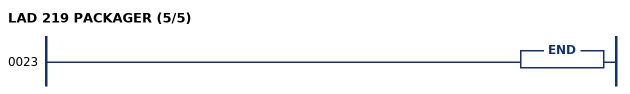
% Rung: 23 %
SOR END EOR

LADDER 220 "NO PACKAGE"
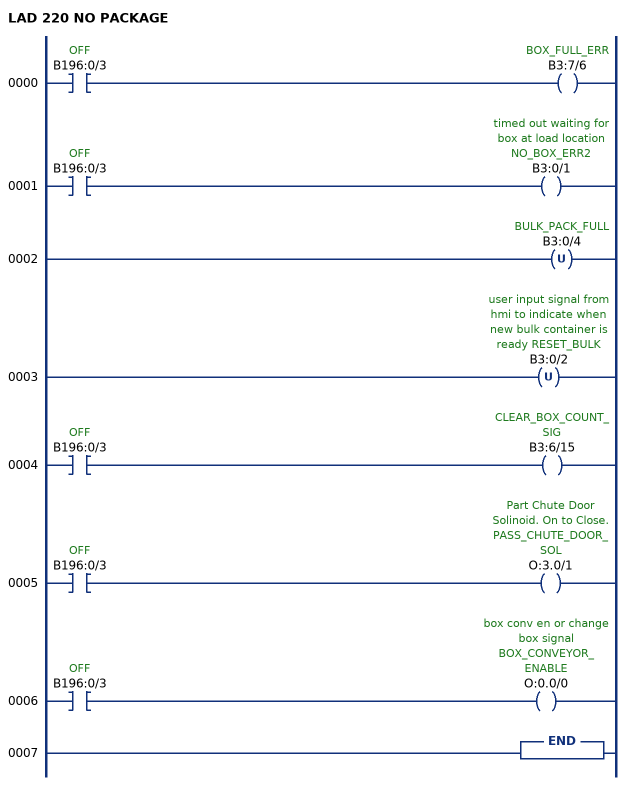
% Rung: 0 %
SOR XIC B196:0/3 OTE B3:7/6 EOR
%   B196:0/3  OFF %
%   B3:7/6  BOX_FULL_ERR %
% Rung: 1 %
SOR XIC B196:0/3 OTE B3:0/1 EOR
%   B196:0/3  OFF %
%   B3:0/1  NO_BOX_ERR2  "timed out waiting for box at load location" %
% Rung: 2 %
SOR OTU B3:0/4 EOR
%   B3:0/4  BULK_PACK_FULL %
% Rung: 3 %
SOR OTU B3:0/2 EOR
%   B3:0/2  RESET_BULK  "user input signal from hmi to indicate when new bulk container is ready" %
% Rung: 4 %
SOR XIC B196:0/3 OTE B3:6/15 EOR
%   B196:0/3  OFF %
%   B3:6/15  CLEAR_BOX_COUNT_SIG %
% Rung: 5 %
SOR XIC B196:0/3 OTE O:3.0/1 EOR
%   B196:0/3  OFF %
%   O:3.0/1  PASS_CHUTE_DOOR_SOL  "Part Chute Door Solinoid. On to Close." %
% Rung: 6 %
SOR XIC B196:0/3 OTE O:0.0/0 EOR
%   B196:0/3  OFF %
%   O:0.0/0  BOX_CONVEYOR_ENABLE  "box conv en or change box signal" %
% Rung: 7 %
SOR END EOR

LADDER 222 "RATE1"
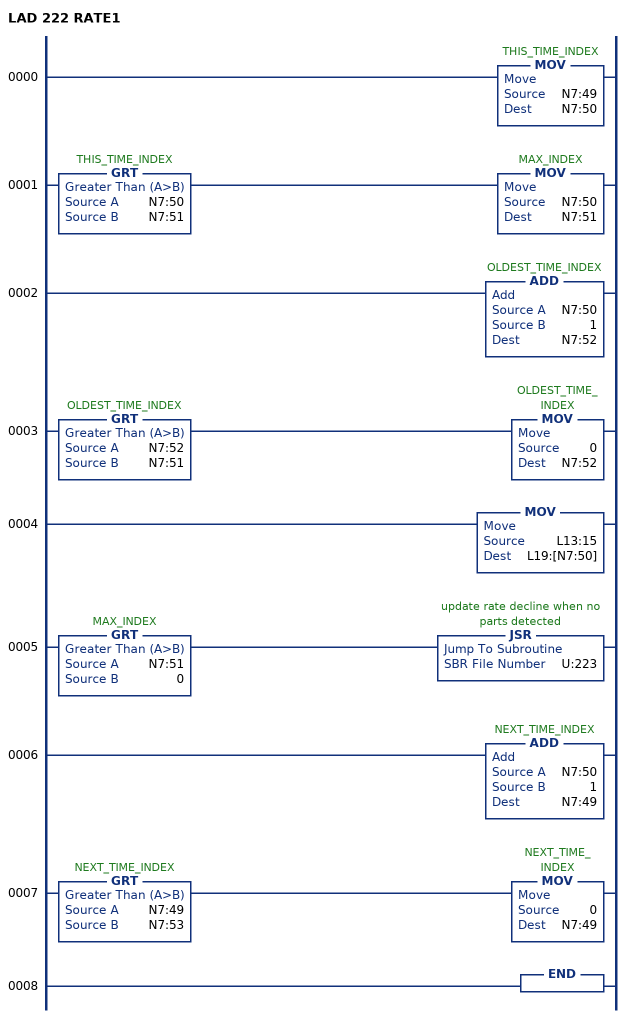
% Rung: 0 %
SOR MOV N7:49 N7:50 EOR
%   N7:49  NEXT_TIME_INDEX %
%   N7:50  THIS_TIME_INDEX %
% Rung: 1 %
SOR GRT N7:50 N7:51 MOV N7:50 N7:51 EOR
%   N7:50  THIS_TIME_INDEX %
%   N7:51  MAX_INDEX %
% Rung: 2 %
SOR ADD N7:50 1 N7:52 EOR
%   N7:50  THIS_TIME_INDEX %
%   N7:52  OLDEST_TIME_INDEX %
% Rung: 3 %
SOR GRT N7:52 N7:51 MOV 0 N7:52 EOR
%   N7:52  OLDEST_TIME_INDEX %
%   N7:51  MAX_INDEX %
% Rung: 4 %
SOR MOV L13:15 L19:[N7:50] EOR
%   L13:15  THE_TIME %
%   N7:50  THIS_TIME_INDEX %
% Rung: 5 %
SOR GRT N7:51 0 JSR U:223 EOR
%   N7:51  MAX_INDEX %
%   U:223  "update rate decline when no parts detected" %
% Rung: 6 %
SOR ADD N7:50 1 N7:49 EOR
%   N7:50  THIS_TIME_INDEX %
%   N7:49  NEXT_TIME_INDEX %
% Rung: 7 %
SOR GRT N7:49 N7:53 MOV 0 N7:49 EOR
%   N7:49  NEXT_TIME_INDEX %
%   N7:53  UPPER_INDEX_LIMIT %
% Rung: 8 %
SOR END EOR

LADDER 223 "RATE2"
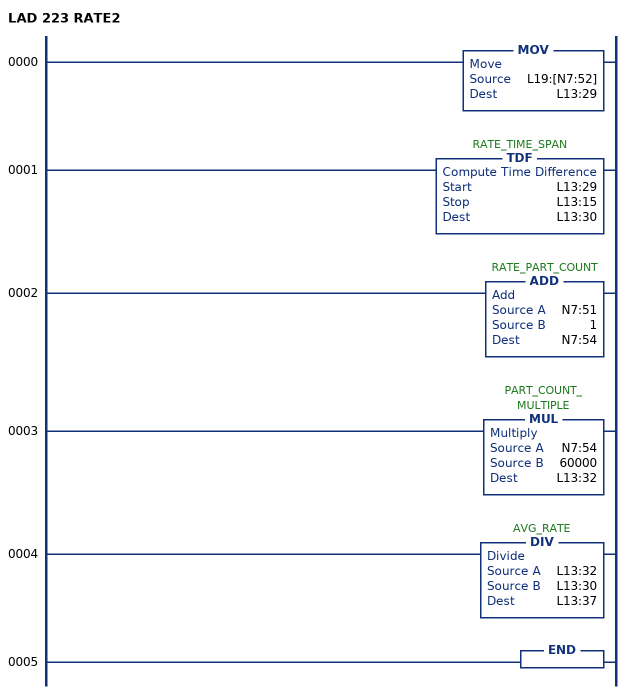
% Rung: 0 %
SOR MOV L19:[N7:52] L13:29 EOR
%   N7:52  OLDEST_TIME_INDEX %
% Rung: 1 %
SOR TDF L13:29 L13:15 L13:30 EOR
%   L13:15  THE_TIME %
%   L13:30  RATE_TIME_SPAN %
% Rung: 2 %
SOR ADD N7:51 1 N7:54 EOR
%   N7:51  MAX_INDEX %
%   N7:54  RATE_PART_COUNT %
% Rung: 3 %
SOR MUL N7:54 60000 L13:32 EOR
%   N7:54  RATE_PART_COUNT %
%   L13:32  PART_COUNT_MULTIPLE %
% Rung: 4 %
SOR DIV L13:32 L13:30 L13:37 EOR
%   L13:32  PART_COUNT_MULTIPLE %
%   L13:30  RATE_TIME_SPAN %
%   L13:37  AVG_RATE %
% Rung: 5 %
SOR END EOR

LADDER 224 "RESET RATE"
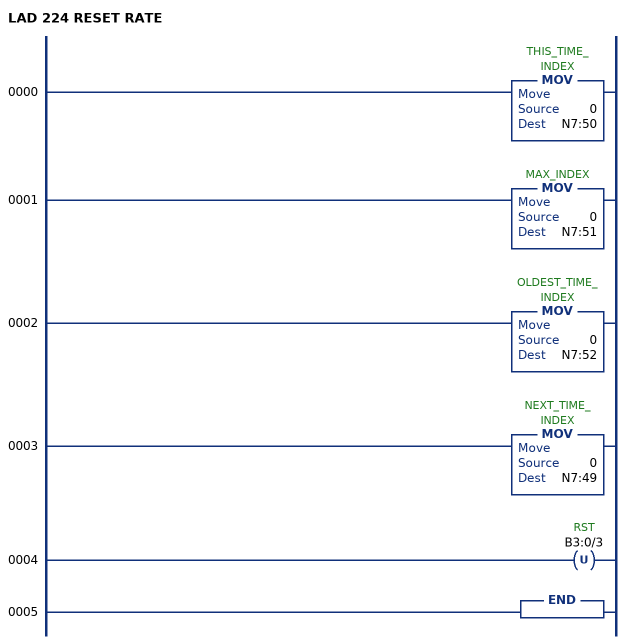
% Rung: 0 %
SOR MOV 0 N7:50 EOR
%   N7:50  THIS_TIME_INDEX %
% Rung: 1 %
SOR MOV 0 N7:51 EOR
%   N7:51  MAX_INDEX %
% Rung: 2 %
SOR MOV 0 N7:52 EOR
%   N7:52  OLDEST_TIME_INDEX %
% Rung: 3 %
SOR MOV 0 N7:49 EOR
%   N7:49  NEXT_TIME_INDEX %
% Rung: 4 %
SOR OTU B3:0/3 EOR
%   B3:0/3  RST %
% Rung: 5 %
SOR END EOR

LADDER 240 "NP STOP"
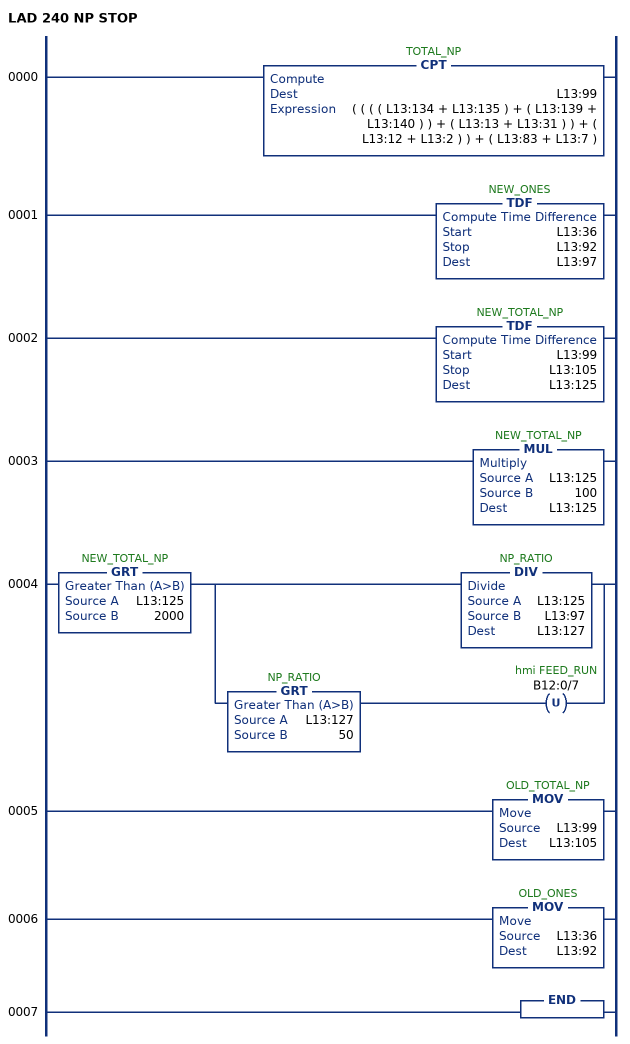
% Rung: 0 %
SOR CPT L13:99 " ( ( ( ( L13:134 + L13:135 ) + ( L13:139 + L13:140 ) ) + ( L13:13 + L13:31 ) ) + ( L13:12 + L13:2 ) ) + ( L13:83 + L13:7 ) " EOR
%   L13:99  TOTAL_NP %
%   L13:134  "too wide bottom" %
%   L13:135  "too close bottom" %
%   L13:139  "too close top count" %
%   L13:140  "too wide top count" %
%   L13:13  SKIP1  "skipped 1 count" %
%   L13:31  SKIP5  "skipped 5 count" %
%   L13:12  SKIP6  "skipped 6 count" %
%   L13:2  INS1_FAIL_COUNT %
%   L13:83  INS5_FAIL_COUNT %
%   L13:7  INS6_FAIL_COUNT %
% Rung: 1 %
SOR TDF L13:36 L13:92 L13:97 EOR
%   L13:36  ONES %
%   L13:92  OLD_ONES %
%   L13:97  NEW_ONES %
% Rung: 2 %
SOR TDF L13:99 L13:105 L13:125 EOR
%   L13:99  TOTAL_NP %
%   L13:105  OLD_TOTAL_NP %
%   L13:125  NEW_TOTAL_NP %
% Rung: 3 %
SOR MUL L13:125 100 L13:125 EOR
%   L13:125  NEW_TOTAL_NP %
% Rung: 4 %
SOR GRT L13:125 2000 BST DIV L13:125 L13:97 L13:127 NXB GRT L13:127 50 OTU B12:0/7 BND EOR
%   L13:125  NEW_TOTAL_NP %
%   L13:97  NEW_ONES %
%   L13:127  NP_RATIO %
%   B12:0/7  FEED_RUN  "hmi" %
% Rung: 5 %
SOR MOV L13:99 L13:105 EOR
%   L13:99  TOTAL_NP %
%   L13:105  OLD_TOTAL_NP %
% Rung: 6 %
SOR MOV L13:36 L13:92 EOR
%   L13:36  ONES %
%   L13:92  OLD_ONES %
% Rung: 7 %
SOR END EOR

LADDER 246 "SPEED BOT"    % high speed %
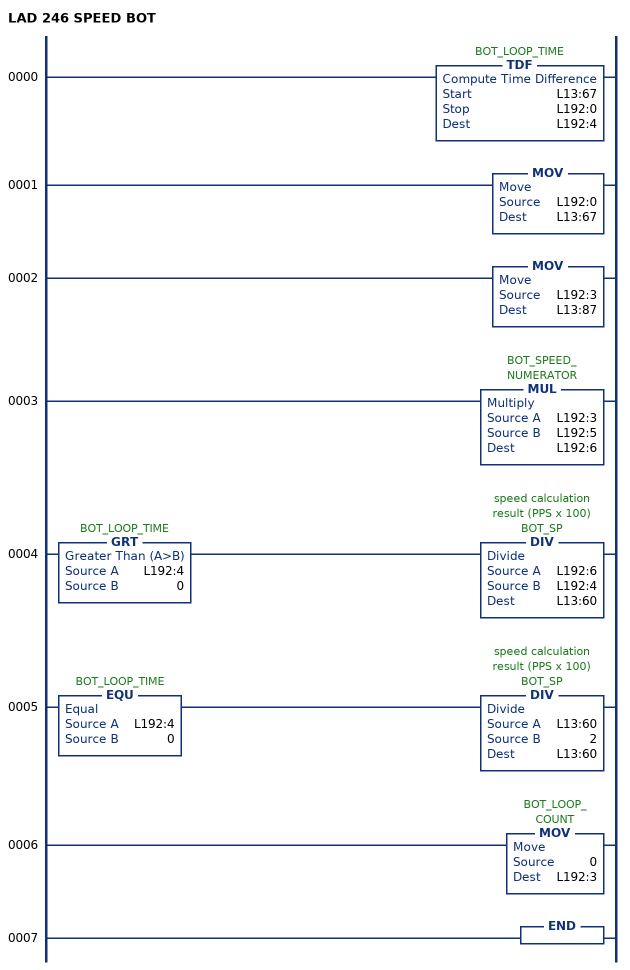
% Rung: 0 %
SOR TDF L13:67 L192:0 L192:4 EOR
%   L192:0  BOT_THIS_TIME  "rtc bot belt movement event time" %
%   L192:4  BOT_LOOP_TIME %
% Rung: 1 %
SOR MOV L192:0 L13:67 EOR
%   L192:0  BOT_THIS_TIME  "rtc bot belt movement event time" %
% Rung: 2 %
SOR MOV L192:3 L13:87 EOR
%   L192:3  BOT_LOOP_COUNT %
% Rung: 3 %
SOR MUL L192:3 L192:5 L192:6 EOR
%   L192:3  BOT_LOOP_COUNT %
%   L192:5  TKS_PER_SECOND %
%   L192:6  BOT_SPEED_NUMERATOR %
% Rung: 4 %
SOR GRT L192:4 0 DIV L192:6 L192:4 L13:60 EOR
%   L192:4  BOT_LOOP_TIME %
%   L192:6  BOT_SPEED_NUMERATOR %
%   L13:60  BOT_SP  "speed calculation result (PPS x 100)" %
% Rung: 5 %
SOR EQU L192:4 0 DIV L13:60 2 L13:60 EOR
%   L192:4  BOT_LOOP_TIME %
%   L13:60  BOT_SP  "speed calculation result (PPS x 100)" %
% Rung: 6 %
SOR MOV 0 L192:3 EOR
%   L192:3  BOT_LOOP_COUNT %
% Rung: 7 %
SOR END EOR

LADDER 248 "SPEED TOP"    % high speed %
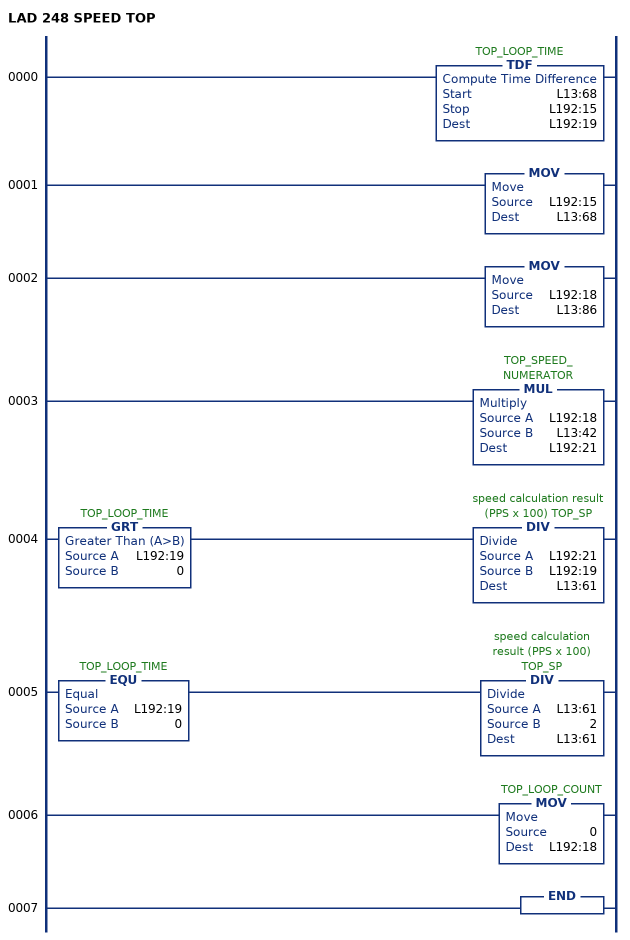
% Rung: 0 %
SOR TDF L13:68 L192:15 L192:19 EOR
%   L192:15  TOP_THIS_TIME  "rtc top belt movement event time" %
%   L192:19  TOP_LOOP_TIME %
% Rung: 1 %
SOR MOV L192:15 L13:68 EOR
%   L192:15  TOP_THIS_TIME  "rtc top belt movement event time" %
% Rung: 2 %
SOR MOV L192:18 L13:86 EOR
%   L192:18  TOP_LOOP_COUNT %
% Rung: 3 %
SOR MUL L192:18 L13:42 L192:21 EOR
%   L192:18  TOP_LOOP_COUNT %
%   L192:21  TOP_SPEED_NUMERATOR %
% Rung: 4 %
SOR GRT L192:19 0 DIV L192:21 L192:19 L13:61 EOR
%   L192:19  TOP_LOOP_TIME %
%   L192:21  TOP_SPEED_NUMERATOR %
%   L13:61  TOP_SP  "speed calculation result (PPS x 100)" %
% Rung: 5 %
SOR EQU L192:19 0 DIV L13:61 2 L13:61 EOR
%   L192:19  TOP_LOOP_TIME %
%   L13:61  TOP_SP  "speed calculation result (PPS x 100)" %
% Rung: 6 %
SOR MOV 0 L192:18 EOR
%   L192:18  TOP_LOOP_COUNT %
% Rung: 7 %
SOR END EOR

LADDER 250 "P BOT"    % high speed %
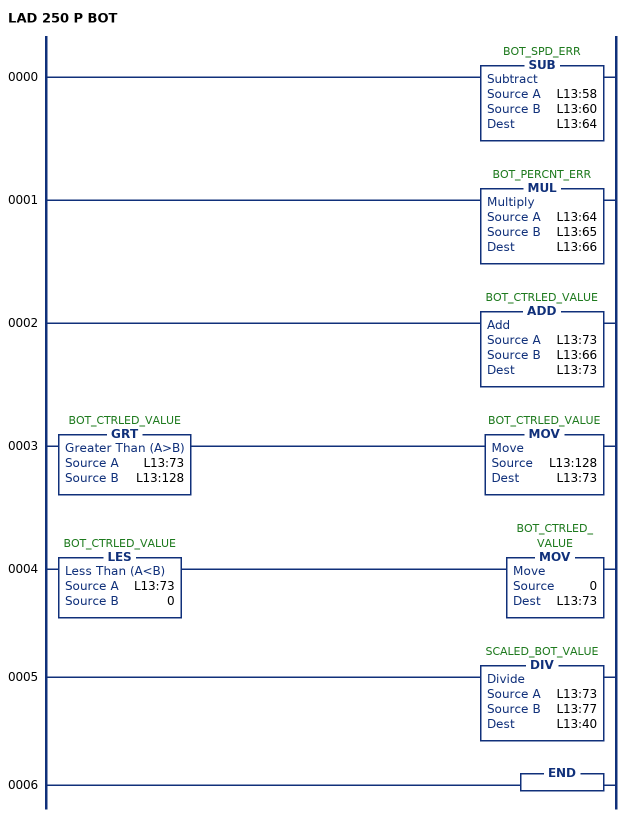
% Rung: 0 %
SOR SUB L13:58 L13:60 L13:64 EOR
%   L13:58  BOT_SPD_SETPOINT %
%   L13:60  BOT_SP  "speed calculation result (PPS x 100)" %
%   L13:64  BOT_SPD_ERR %
% Rung: 1 %
SOR MUL L13:64 L13:65 L13:66 EOR
%   L13:64  BOT_SPD_ERR %
%   L13:65  POS5SHIFT %
%   L13:66  BOT_PERCNT_ERR %
% Rung: 2 %
SOR ADD L13:73 L13:66 L13:73 EOR
%   L13:73  BOT_CTRLED_VALUE %
%   L13:66  BOT_PERCNT_ERR %
% Rung: 3 %
SOR GRT L13:73 L13:128 MOV L13:128 L13:73 EOR
%   L13:73  BOT_CTRLED_VALUE %
%   L13:128  "how much top has shifted since measurment" %
% Rung: 4 %
SOR LES L13:73 0 MOV 0 L13:73 EOR
%   L13:73  BOT_CTRLED_VALUE %
% Rung: 5 %
SOR DIV L13:73 L13:77 L13:40 EOR
%   L13:73  BOT_CTRLED_VALUE %
%   L13:40  SCALED_BOT_VALUE %
% Rung: 6 %
SOR END EOR

LADDER 252 "P TOP"    % high speed %
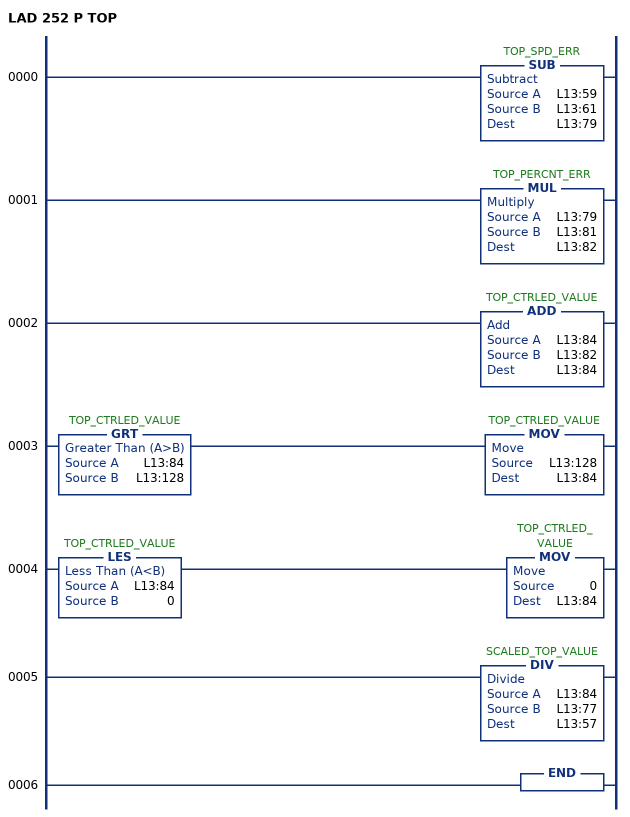
% Rung: 0 %
SOR SUB L13:59 L13:61 L13:79 EOR
%   L13:59  TOP_SPD_SETPOINT %
%   L13:61  TOP_SP  "speed calculation result (PPS x 100)" %
%   L13:79  TOP_SPD_ERR %
% Rung: 1 %
SOR MUL L13:79 L13:81 L13:82 EOR
%   L13:79  TOP_SPD_ERR %
%   L13:81  TOP_FDBK_RATIO %
%   L13:82  TOP_PERCNT_ERR %
% Rung: 2 %
SOR ADD L13:84 L13:82 L13:84 EOR
%   L13:84  TOP_CTRLED_VALUE %
%   L13:82  TOP_PERCNT_ERR %
% Rung: 3 %
SOR GRT L13:84 L13:128 MOV L13:128 L13:84 EOR
%   L13:84  TOP_CTRLED_VALUE %
%   L13:128  "how much top has shifted since measurment" %
% Rung: 4 %
SOR LES L13:84 0 MOV 0 L13:84 EOR
%   L13:84  TOP_CTRLED_VALUE %
% Rung: 5 %
SOR DIV L13:84 L13:77 L13:57 EOR
%   L13:84  TOP_CTRLED_VALUE %
%   L13:57  SCALED_TOP_VALUE %
% Rung: 6 %
SOR END EOR

LADDER 254 "TOTALCOUNT"
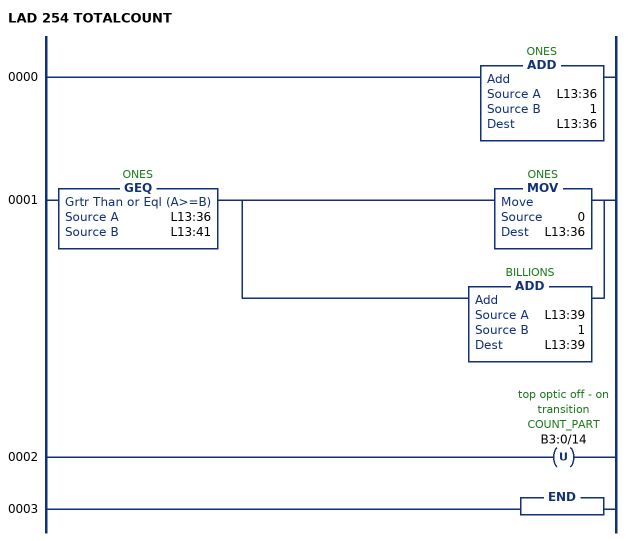
% Rung: 0 %
SOR ADD L13:36 1 L13:36 EOR
%   L13:36  ONES %
% Rung: 1 %
SOR GEQ L13:36 L13:41 BST MOV 0 L13:36 NXB ADD L13:39 1 L13:39 BND EOR
%   L13:36  ONES %
%   L13:41  "skipped count change in the last 3 seconds" %
%   L13:39  BILLIONS %
% Rung: 2 %
SOR OTU B3:0/14 EOR
%   B3:0/14  COUNT_PART  "top optic off - on transition" %
% Rung: 3 %
SOR END EOR

OTHER DOCUMENTED ADDRESSES
  B3:1/14  ALIGNMENT_OK
  B3:6/12  "turn off to block triggers after above time"
  B3:10/14  "Dont use"
  B38:0  EX1_GOOD
  B40:0  EX3_GOOD
  B189:0/0  "change box"
  B189:0/9  "override boxing ok or not full signal"
  B189:0/11  "HMI force door close"
  B196:1/0  "Chute door is closed"
  B196:1/1  "control chute door"
  B196:1/13  "force box conveyor on"
  B196:3/0  "for hmi to continue production unlatched by hmi"
  BUL_COUNT_REACHED  
  F8:5  PPM_AVG_F
  F8:98  "time in multiples of 10 us"
  F8:99  "loop time in milliseconds"
  F193:6  BOT_FDBK_RATIO
  F193:14  SCALED_TOP_SETPOINT
  HSC:0.0  "top"
  HSC:0.3/6  "Underflow interrupt"
  HSC:0.3/7  "Overflow interrupt"
  HSC:1.0  "bot"
  HSC:1.3/6  "Underflow interrupt"
  HSC:1.3/7  "Overflow interrupt"
  I:0.0/0  "Encoder Signal "A""
  I:0.0/1  "Encoder Signal "B""
  I:0.0/3  CHUTE_OPTIC_2
  I:0.0/4  "Encoder Signal "A""
  I:0.0/5  "Encoder Signal "B""
  I:0.0/11  PASS_4
  I:0.0/15  ACQ_4
  I:0.1/3  FAIL_4
  I:0.1/4  "not used"
  I:0.1/5  "not used"
  I:0.1/6  "not used"
  I:0.1/7  "not used"
  I:0.1/8  "not used"
  I:0.1/9  "not used"
  I:0.1/10  "not used"
  I:0.1/11  "not used"
  I:0.1/12  "not used"
  I:0.1/13  "not used"
  I:0.1/14  "not used"
  I:0.1/15  "not used"
  I:0.2  "not used"
  I:0.2/3  "Packaging Conveyor full"
  I:0.2/4  "Packaging Conveyor Box in Position"
  I:0.3  "not used"
  I:0.4  "Spare Analog Input 1"
  I:0.5  "Spare Analog Input 2"
  I:0.6  "Spare Analog Input 3"
  I:2.0/0  FRONT_ESTOP
  I:2.0/1  REAR_ESTOP
  I:2.0/8  FRONT_DOOR  "front door signal ce models only"
  I:2.0/9  REAR_DOOR  "rear door signal ce models only"
  I:2.0/10  MAINTENANCE_KEY_SW  "Maintenance Key Switch ce models only"
  I:2.0/11  "spare"
  I:2.0/12  "spare"
  I:2.0/14  "spare"
  L13:130  "virtual part to real part offset"
  L13:138  "alignment fail counts"
  L13:145  "times processed"
  L13:146  "times processed good"
  L13:147  "1/2 of times processed"
  L13:157  "I2 Avg queue over peak limit count"
  L13:160  "I2 Avg queue over timed limit count"
  L13:162  "I2 Max queue"
  L13:163  "I2 Max avg queue"
  L13:164  "I2 Max acq time"
  L13:165  "I1 Max Queue"
  L13:166  "I1 Maximum avg queue"
  L13:167  "I1 Avg queue over peak limit count"
  L13:168  "I1 Avg queue over timed limit count"
  L13:170  "I1 Max acq time"
  L13:171  "max process 1 time"
  L13:172  "max process 5 time"
  L13:173  "max process 6 time"
  L13:180  "maximum time between triggers"
  L13:181  "minimum okay time between triggers"
  L13:182  RATE_QUEUE_LIMIT
  L13:184  "intermediate i1 trig avg"
  L13:185  I1_TBT  "i1 average time between triggers"
  L13:186  "intermediate i5 trig avg"
  L13:187  I5_TBT  "i5 average time between triggers"
  L13:188  "intermediate i6 trig avg"
  L13:189  I6_TBT  "i6 average time between triggers"
  L13:190  "i1 timed q limit"
  L13:191  "i1 absolute q limit"
  L16:2  TRIG_DELAY_Q_MULTI
  L16:3  TRIG_DELAY_MIN_TIME
  L16:4  TRIG_DELAY_FLAT_RATE
  L16:5  CLEARTIME1  "time to clear tracking data"
  L16:6  CLEARTIME5
  L16:7  CLEARTIME6
  L16:8  PASS1PRTLOC
  L16:9  PASS1PROCESSTM
  L16:11  PASS5PROCESSTM
  L16:13  PASS6PROCESSTM
  L23:19  TOP_OPT_FAIL_CT
  L23:34  AIR_PRESSURE_FAULT
  L28:0  INS_1_TIME
  L29:0  INS_1_POS
  L30:0  INS_5_TIME
  L31:0  INS_5_POS
  L32:0  INS_6_TIME
  L33:0  INS_6_POS
  L183:2  "simulated part width"
  L183:3  "button state"
  L183:5  TFTT1  "timer count for test trigger 1"
  L183:6  TFTT5  "timer count for test trigger 5"
  L183:7  TFTT6  "timer count for test trigger 6"
  L187:0  ACQTM1
  L187:1  ACQTM5
  L187:2  ACQTM6
  L187:5  "pass transfer out signals"
  L187:6  "NoErr transfer out signals"
  L187:7  "ins 1 trigger count"
  L190:1  "count of gap fails"
  L190:2  "I1 blocked triggers"
  L190:4  "count of parts rejected because acquire time ran out"
  L190:5  "count of parts that received a pass signal but previously failed 1"
  L190:6  "count of result signals received with no part present 1"
  L190:7  "count of results received after maximim time reached"
  L190:8  "pass count"
  L190:9  "fail count"
  L190:10  "acquisition count"
  L190:11  "acquisition without result count"
  L190:12  "count of parts results that time out"
  L190:27  "optic alignment pass signal"
  L190:28  "optic alignment fail signal"
  L190:31  "something wrong, can't happen"
  L190:32  "Crazy wrong, can't happen"
  L192:1  BOT_LAST_TIME  "rtc bot belt previous movement event time"
  L192:2  BOT_CYCLE_TIME  "rtc bot belt time between events"
  L192:7  FROM_REAL  "distance from real part signal at optic location"
  L192:8  FROM_TRACKED  "distance from tracked part signal at optic location"
  L192:16  TOP_LAST_TIME  "rtc top belt previous movement event time"
  L192:17  TOP_CYCLE_TIME  "rtc top belt time between events"
  L199:5  ACQTM51
  L199:6  ACQTM52
  L199:7  ACQTM53
  L199:9  "ones"
  L199:10  "billions"
  L199:13  DUMP_LONG
  L199:15  ACQTM11
  L199:16  ACQTM12
  L199:17  ACQTM13
  L199:20  RESULTTM1
  L199:22  CLEARTIME5COUNT
  L199:23  CLEARTIME6COUNT
  L199:24  ACQTM61
  L199:25  ACQTM62
  L199:26  ACQTM63
  L199:27  TMSINCETRIG1
  L199:29  TMSINCETRIG5
  L199:30  TMSINCETRIG6
  L199:31  CLEARTIME1COUNT
  L199:32  RESULTTM5
  L199:33  RESULTTM6
  L199:34  MAXACQTM1
  L199:36  MAXACQTM6
  L201:1  CAM_5_MIN_CY
  L201:2  CAM_6_MIN_CY
  L201:5  "ms since trig 1 is initialized"
  L201:10  "movement from virtual (pos, add)"
  L204:1  TTT5
  L204:2  TTT6
  L204:3  "last time between ins 5 triggers"
  L204:7  "last trigger to trigger time"
  L204:13  "This optic signal time"
  L204:14  "Last optic signal time"
  L204:15  "time between optic signals"
  N10:1  "old ConveyorStatus"
  N10:2  "PowerOn"
  N10:3  "Local Mode On BypassBoxingPLC"
  N10:4  "Boxing Connected Signal"
  N10:5  "BoxJamSignal"
  N10:6  "WaittingOnBoxSig"
  N10:7  "ConveyorFullSig"
  N10:8  "MachineFaultSig"
  N10:9  "Counter Sensor Fault"
  N10:11  "Feeder Track Sensor Blocked"
  N10:12  "Air Pressure Fault"
  N13:0  "Part Inspecting"
  N13:4  "Completed Counter"
  N13:5  "Trigger Position Counter"
  N13:6  "BlowOff Start Counter"
  N13:7  "BlowOff Stop Counter"
  N13:8  "Inspection Command Counter"
  N13:9  "Complete Counter"
  N13:10  "Pass Signal Counter"
  N13:11  "Solenoid Signal Counter"
  N13:12  "Hold Pass Counter"
  N13:13  "Hold Pass Length"
  N16:1  "Bottom Inspection Offset For Tracking"
  N16:3  "Bit Shift Preset"
  N17:5  "Parts In Tube Counter"
  N17:6  "Parts In Tube Limit"
  N17:9  "Bot to Top Transfer Position"
  N17:12  "Trigger to laser Counter"
  N197:1  "maximim acquire time 1"
  N197:2  "time for chute door to close"
  N197:3  "FeedWheel Speed Output Setting"
  N197:4  "boxing convery full time out time (ms)"
  N197:5  "Feeder Speed Output Setting"
  N197:10  "pulse distance to keep blow on then turn off feed"
  N197:11  "speed in pps"
  N197:12  "seconds of ontime"
  N197:20/0  "Deformed Head Blowoff Bit to TOP PLC"
  N200:1  RESULTPOS6B
  N200:2  RESULTPOS5A
  N200:3  RESULTPOS5B
  N200:4  RESULTPOS5C
  N200:5  DUMP_INT
  N200:6  PLATOL  "part location at top optic load"
  N200:7  RESULTPOS5D
  N200:8  RESULTPOS6C
  N200:9  RESULTPOS6D
  N200:10  ACQPOS11
  N200:11  ACQPOS12
  N200:12  ACQPOS13
  N200:14  ACQPOS1  "part acq pos 1"
  N200:15  RESULTPOS1  "result position 1"
  N200:17  RESULTPOS5
  N200:18  RESULTPOS6
  N200:19  ACQPOS5  "part acq pos 5"
  N200:20  ACQPOS6  "part acq pos 6"
  N200:21  ACQPOS51
  N200:22  ACQPOS52
  N200:23  ACQPOS53
  N200:24  ACQPOS61
  N200:25  ACQPOS62
  N200:26  ACQPOS63
  O:0.0/1  "spare"
  O:0.0/5  INS_4_TRIG
  O:0.0/6  "spare"
  O:0.0/10  FEED_WHEEL_EN
  O:0.0/11  "Spare"
  O:0.0/12  "not used"
  O:0.0/13  "not used"
  O:0.0/14  "not used"
  O:0.0/15  "not used"
  O:0.1  "not used"
  O:0.2  "not used"
  O:0.3  "not used"
  O:0.5  "spare analog output"
  O:3.0/0  "spare"
  O:3.0/2  "spare"
  O:3.0/3  "light curtain range selection /* needed? */"
  O:3.0/7  "door unlocks on CE models"
  O:3.0/8  "spare"
  O:3.0/9  "spare"
  O:3.0/10  "spare"
  PFILE:6  "check for part jams"
  PFILE:10  "Bottom belt HSC"
  PFILE:12  "Top belt HSC"
  Q2:55  END_OF_MAIN
  Q5:94  END_OF_BELTS
  R6:2  "track part location until acquire 5"
  R6:3  "track acquire time 5"
  R6:5.POS  "Empty Fifo"
  R6:8  "track part location until acquire 6"
  R6:9  "track acquire time 6"
  R21:0  "Trigger Shift Register"
  T20:0  "Trigger On Time"
  U:9  "slow data"
  U:11  "transfered data calcuations from the high speed section"
  U:24  "check skipped fail rate"
  U:28  "faults"
  U:29  "speed"
  U:30  "count"
  U:31  "rate calc"
  U:32  "boxer"
  U:33  "bulk pack"
  U:34  "customer boxing unit signals"
  U:35  "cleanup"
  U:180  "rate calc"

COMMENTS NOT ATTACHED TO A CURRENT RUNG
  F8:13: *************************
    Loads Side Camera Passing data into a bit shift
    *************************
    
    loads passing data bit into passing data bit shift register at the part present cl.
  I:0.0/8: special rung for testing. This rung can simulate a pass signal. It will not be timed correctly.
  B23:0/0: Yet another bit shift load with data in the part position indicating that there was a bottom system part pass as well as a top system part present at this location.
    
    verified works w/bypassed 071910 and unbypassed 072010
  N7:25: 1050
  C5:4: tempory counting to verify pass part count with boxing part count.
  B22:0/0: ***********************
     Bottom Part Syncronizing Logic
    ***********************
    
    This is the point at the bottom of the top conveyor where the part jumps from the bottom conveyor.  This system will then track the part through the top system to the point of the laser optic in order to verify that the part in question has passed the bottom inspection.  I believe that we NEED to include FAILING inspections to eliminate the possibility of a out of position part from passing. LW 072010
  T20:2.ACC: This rung is starting a timer that should be activated directly before the laser optic part presense sensor on the top conveyer and should cause the top optic to be ignored if the bottom camera system didn't pass. however other arrangements must be made if the bottom camera isn't going to be used as is the case with a nut inspection.
  T20:2: The timer used to verify that the part that triggered the top laser optic has passed the bottom camer. needs to be count
  N17:8: ****************************************************************************************************************
    I can not find anywhere in the program where the "Test Spacing From Pickup to Trigger is activated indicating to me that this entire function must not be doing anything in this program at this time.
    ****************************************************************************************************************
  B11:0/0: load part present bit shit with one shot data from the part present sensor
  B3:6/1: ***********************
    Part Width and  Location
    ***********************
    
    Calculates the position of parts on the top belt by measureing the part width by calculating the number of belt movement pulses that occure when the optic is blocked and then devides that in half and add that to the optic location in the part presnet bit shift when the top optic is cleared.
  N7:45: not fully functional because of part overlap but measurems the camera responce time when part inspections are not overlaping
  B9:0/[N7:47]: Remove any part present signals outside of expected location
  B9:0/[N7:50]: Remove any part present signals outside of expected location
  F19:0: Counter inside of a high speed counter interrupt counts the number of Bit Shifts that need to be processed in order to move the logic with the parts on the conveyor.
  F8:14: **************
    Bottom Top Camera Trigger
    *************
    
    Trigger Bottom Top Camera
  N10:4: test if boxing is connected
  B3:11/3: After initial delay allow blow two start functioning
  T4:28: Check for buffer reset
  RUNG000150-000011: trigger count
  RUNG000150-000012: wipe stored part data if acq time expires
  RUNG000150-000013: clear data for aquire time expired
  RUNG000150-000014: clear data for time
  RUNG000150-000016: wiped count
  RUNG000150-000018: pass, fail and acquire inputs
  RUNG000150-000025: pass code / Set pass bit in Bit Shift
    captures result position and processing time
    Unlatch pass bit
  RUNG000150-000032: pass count
  RUNG000150-000035: fail count
  RUNG000150-000038: acquire code
  RUNG000150-000039: Grab trigger/acquire position
    Grab acquire time
  RUNG000150-000041: transfer tracked part positon from trigger/acquire to the acquire/result
    capture acquire time
    reset process time
  L14:8: on when ok for run
  L14:3: off when ok to run
  L14:2: off when ok to run
  L14:5: on when ok to run, rear off turns both off
  L13:165: maximum q i1
  N7:76: removed relieance on trigger signal
  N197:20/0: Passes deformed head blowoff command to TOP PLC where solenoid output is located.
  L13:162: maximum q
  L13:163: maximum average q
  N7:47: ***********************************************************************************************************************************************************
    From side
    ***********************************************************************************************************************************************************
    
    removed relieance on trigger signal
  B3:10/1: prevents momentary signals from box present sensor from tripping the logic for box not present
    
    This is in responce to a problem created by the sensor occasionally turning on as if no box was in its path when there is a box present.
  B3:6/2: IF PROCESSING FAULT OCURES AT COUNTER SENSOR; CLEAR THE BELT OF PASSING DATA
  L14:23: ****************  nEEDS fIXING  **********************
  L14:36: ****************  nEEDS fIXING  **********************
  RUNG000010-000014: ****
                      Zeros out the non passing part count when one passes
    ****
  RUNG000010-000018: Remove any part present signals outside of expected location
  T4:27: Check for buffer reset
  T4:26: Check for buffer reset
  RUNG000125-000014: clear data for time
  RUNG000125-000013: clear data for aquire time expired
  RUNG000125-000012: wipe stored part data if acq time expires
  RUNG000125-000011: trigger count
  RUNG000125-000029: Set pass bit in Bit Shift
    captures result position and processing time
    Unlatch pass bit
  RUNG000125-000027: transfer tracked part positon from trigger/acquire to the acquire/result
    capture acquire time
    reset process time
  RUNG000125-000026: Grab trigger/acquire position
    Grab acquire time
  RUNG000125-000025: pass code / Set pass bit in Bit Shift
    captures result position and processing time
    Unlatch pass bit
  RUNG000125-000018: pass, fail and acquire inputs
  RUNG000125-000016: wiped count

REVISION NOTES
  13: updated count reset
  14: added io moduals
  15: multiple steps toward new hmi integration
  21: test

DATA TABLE (non-zero values as saved)
DATA B3
% B3:0 % 0XA020 0X0000 0X4005 0XA000 0X5E7D 0X0560 0X0622 0X0421 0X4006 0X0000
% B3:10 % 0X2041 0X0846 0X2000 0X0000
DATA T4
% .PRE .ACC %
% T4:0 % 0 2
% T4:1 % 150 0
% T4:2 % 400 0
% T4:3 % 333 118
% T4:4 % 300 300
% T4:5 % 250 0
% T4:6 % 10 32766
% T4:7 % 666 0
% T4:8 % 20 0
% T4:9 % 50 43
% T4:10 % 200 200
% T4:11 % 3333 0
% T4:12 % 35 40
% T4:13 % 250 0
% T4:14 % 666 0
% T4:15 % 150 0
% T4:16 % 11 0
% T4:17 % 100 59
% T4:18 % 120 120
% T4:19 % 300 0
% T4:20 % 200 0
% T4:21 % 200 0
% T4:22 % 200 0
% T4:23 % 250 0
% T4:24 % 666 0
% T4:25 % 50 0
% T4:26 % 250 0
% T4:27 % 250 0
% T4:28 % 250 0
% T4:29 % 5000 0
% T4:30 % 333 116
% T4:31 % 333 110
% T4:32 % 69 0
DATA C5
% .PRE .ACC %
% C5:0 % 32766 0
DATA R6
% .LEN .POS %
% R6:0 % 1250 0
% R6:1 % 1250 0
% R6:2 % 3 0
% R6:3 % 3 0
% R6:4 % 1250 0
% R6:5 % 1250 0
% R6:6 % 1250 0
% R6:7 % 10 0
% R6:8 % 3 0
% R6:9 % 3 0
% R6:10 % 2000 0
% R6:11 % 1024 0
% R6:12 % 10 0
% R6:13 % 10 0
% R6:14 % 10 0
% R6:15 % 10 0
% R6:16 % 1250 0
% R6:17 % 2000 0
% R6:18 % 1024 0
% R6:19 % 10 0
DATA N7
% N7:0 % 32767 3 1051 300 300 400 0 32767 500 500
% N7:10 % 1000 61 0 2 20 20 1000 2000 50 1050
% N7:20 % 32767 333 10 333 333 46 19 0 19 250
% N7:30 % 666 32767 150 0 0 102 6 49 0 49
% N7:40 % 0 41 0 41 1242 1520 1251 1555 5 3
% N7:50 % 2 16 3 16 17 32766 32766 0 32766 0
% N7:60 % 1250 2000 1024 1052 1026 1016 0 15 30 20
% N7:70 % 0 21 23 27738 32767 0 122 0 16 0
% N7:80 % 0 6 95 0 0 0 5 500 0 0
% N7:90 % 2011 4 4 12 1 0 0 0 0 1600
% N7:100 % 1003 90 110 100 175 25 0 0 0 0
DATA F8
% F8:0 % 0 1 23807 499 0.23807
% F8:5 % 0 0 500 1.9 2
% F8:10 % 1 0.08897486 3058 101 63.26563
% F8:15 % 37.73437 4040 2 0 0
% F8:20 % 0 0.02 0 1 0
% F8:25 % 0 932781 0.222 279.6551 848597
% F8:30 % 0 170 0.03 38 852060
% F8:35 % 0 0 0 0 77
% F8:40 % 101 37.73437 0 100 1
% F8:45 % 1 2 0.21455 0 0
% F8:50 % 0 0 1 0 1
% F8:55 % 2000000 -221 0 0 0
% F8:95 % 0 0 0 492 4.92
DATA B12
% B12:0 % 0X0144 0X0000 0X0000 0X0000 0X0000 0X0000 0X0000 0X0000 0X0000 0X0000
DATA L13
% L13:0 % 4670163 0 0 78522801 283500250
% L13:5 % 4727 0 0 1545317 72789
% L13:10 % 633923782 0 0 0 25
% L13:15 % 285114481 -2147483648 2147483647 2147483647 82058
% L13:20 % 638754657 639611381 777 633923782 100
% L13:25 % 2147483647 25 29503 0 285008542
% L13:30 % 105042 429 1020000 285066205 444
% L13:35 % 12149 5966 10 0 0
% L13:40 % 4284 1000000000 1000000 285066177 0
% L13:45 % 60 700 0 28 639608946
% L13:50 % 0 48347 220636856 0 60
% L13:55 % 0 650 2957 500 500
% L13:60 % 498 498 28 800 2
% L13:65 % 100 200 1444792389 1444792755 204977487
% L13:70 % 638464282 23 22 428400 639608946
% L13:75 % 2 0 100 220636879 2
% L13:80 % 23 74 148 0 295741
% L13:85 % 2627 26 26 26483 1000
% L13:90 % 26616 0 5966 1000 0
% L13:95 % 60 3372 0 25989 439
% L13:100 % 2200 1 2100 3 664
% L13:105 % 439 21 638554790 58 638554785
% L13:110 % 5 30 0 639608757 639608748
% L13:115 % 639608757 9 5 639608752 1100
% L13:120 % 1 170 10 30 215
% L13:125 % 0 638464282 2147483647 3276500 2629
% L13:130 % -2 2 -2 -2 0
% L13:135 % 0 1000 2629 12 8
% L13:140 % 2 11 36 50 50
% L13:145 % 2124371 22465 1284 0 100
% L13:150 % 12 20 170 -170 0
% L13:155 % 0 -8 24 0 2180
% L13:160 % 3 7 4 395082 53203921
% L13:165 % 3 189116 95 13 8150
% L13:170 % 55946610 30 72 54 0
% L13:175 % 0 0 42 23 38
% L13:180 % 176247033 25 99000 52866 644409
% L13:185 % 64 916459 92 627156 63
% L13:190 % 4 5 0 0 0
DATA F14
% F14:0 % 1.32889e-38 5747.126 1550 1550 1638.3
% F14:5 % 1638.3 1638.3 1638.3 0 0
DATA N15
% N15:0 % 6 950 1500 1250 1240 111 100 1172 1046 10
% N15:10 % 65 460 0 0 0 0 1172 0 0 0
DATA L16
% L16:0 % 8 35 11 0 20
% L16:5 % 250 5000 5000 182 19
% L16:10 % 1256 18 2045 6599584 98
% L16:15 % 99 0 0 0 0
DATA L19
% L19:0 % 285055678 285059052 285062429 285008542 285011983
% L19:5 % 285015396 285018795 285022199 285025609 285029010
% L19:10 % 285032082 285035380 285038788 285042165 285045541
% L19:15 % 285048910 285052305 0 0 0
DATA L28
% L28:0 % 201306404 201326824 201385582 201410930 202463998
% L28:5 % 202464202 204294884 204406189 204425660 204461808
% L28:10 % 204508848 204596228 204975419 204975759 204976100
% L28:15 % 204976441 204976781 204977121 204977462 283500250
% L28:20 % 104320977 104344931 131290028 131314625 131364897
% L28:25 % 131365149 131382028 131382331 131398557 131399025
% L28:30 % 131416570 131416931 131434034 131434222 195668988
% L28:35 % 195688241 195703502 195719096 195782688 195838867
% L28:40 % 195904932 195911863 195939739 195940000 195978078
% L28:45 % 195978474 196028235 196028514 201254185 201296964
DATA L29
% L29:0 % 633108849 633113377 633126410 633132031 633365572
% L29:5 % 633365617 633771626 633796313 633800631 633808650
% L29:10 % 633819082 633838460 633922637 633922783 633922950
% L29:15 % 633923137 633923340 633923555 633923782 638593928
% L29:20 % 619325237 619330549 625306226 625311681 625322828
% L29:25 % 625322884 625326627 625326694 625330291 625330395
% L29:30 % 625334286 625334366 625338159 625338201 631858627
% L29:35 % 631862897 631866281 631869739 631883840 631896298
% L29:40 % 631910950 631912487 631918669 631918727 631927171
% L29:45 % 631927259 631938295 631938357 633097269 633106756
DATA L30
% L30:0 % 284902318 284905724 284909133 284912538 284915951
% L30:5 % 284919355 284922764 284926166 284929574 284932977
% L30:10 % 284936380 284939791 284943193 284946604 284950007
% L30:15 % 284953410 284956860 284960255 284963667 284967113
% L30:20 % 284970514 284973924 284977328 284980733 284984141
% L30:25 % 284987548 284990952 284994360 284997764 285001173
% L30:30 % 285004575 285007984 285011383 285014796 285018233
% L30:35 % 285021635 285025045 285028446 285031488 285033592
% L30:40 % 285035764 285039102 285042542 285045914 285049287
% L30:45 % 285052661 285056054 285059428 285062805 285066177
DATA L31
% L31:0 % 639603280 639603383 639603486 639603589 639603692
% L31:5 % 639603795 639603898 639604001 639604104 639604207
% L31:10 % 639604310 639604413 639604516 639604619 639604722
% L31:15 % 639604825 639604929 639605032 639605135 639605239
% L31:20 % 639605342 639605445 639605548 639605651 639605754
% L31:25 % 639605857 639605960 639606063 639606166 639606269
% L31:30 % 639606372 639606475 639606578 639606681 639606785
% L31:35 % 639606888 639606991 639607094 639607197 639607300
% L31:40 % 639607413 639607582 639607755 639607925 639608095
% L31:45 % 639608265 639608436 639608606 639608776 639608946
DATA L32
% L32:0 % 220582818 220583510 220584201 220584893 220585590
% L32:5 % 220586285 220586977 220587672 220588368 220589063
% L32:10 % 220589760 220590455 220591146 220591842 220592544
% L32:15 % 220593233 220593923 220594612 220595308 220596004
% L32:20 % 220596693 220597387 220598084 220598783 220599479
% L32:25 % 220600174 220600868 220601564 220602256 220602945
% L32:30 % 220603638 220604331 220605029 220605074 220632176
% L32:35 % 220632988 220633661 220634294 220634920 220635550
% L32:40 % 220636192 220636856 220578675 220579330 220580029
% L32:45 % 220580073 220580721 220581418 220581463 220582116
DATA L33
% L33:0 % 638463715 638463729 638463743 638463757 638463771
% L33:5 % 638463785 638463799 638463813 638463827 638463841
% L33:10 % 638463855 638463869 638463883 638463897 638463911
% L33:15 % 638463925 638463939 638463952 638463967 638463981
% L33:20 % 638463995 638464009 638464023 638464037 638464051
% L33:25 % 638464065 638464079 638464093 638464107 638464121
% L33:30 % 638464135 638464148 638464163 638464163 638464186
% L33:35 % 638464201 638464215 638464229 638464242 638464255
% L33:40 % 638464268 638464282 638463631 638463644 638463659
% L33:45 % 638463659 638463673 638463687 638463687 638463701
DATA B35
% B35:70 % 0X0000 0X0000 0X0000 0X0000 0X0000 0X0000 0X0000 0X0000 0X0000 0XFFFF
% B35:80 % 0XFFFF 0XFFFF 0X611F 0X4080 0X007F 0X0000 0X0000 0X0000 0X0000 0X0000
DATA L192
% L192:0 % 1444961925 266932201 5055 9 49848
% L192:5 % 1000000 25000000 999 999 8
% L192:10 % 0 0 0 78 17
% L192:15 % 1444962835 332250347 860888 9 51955
% L192:20 % 180 26000000 0 0 0
DATA B196
% B196:0 % 0X0815 0X9FFE 0X0005 0X0000 0X0000 0X0000 0X0000 0X0000 0X0000 0X0000
% B196:30 % 0XE800 0X9BFF 0XEBFF 0XFFDF 0XFFFF 0X0000 0X0000 0X0000 0X0000 0X0000
DATA L199
% L199:0 % 1 0 0 0 0
